INTERFACE ITF_SubSystem

PROPERTY PUBLIC eCondition : SubLevelCondition
GET
END_GET
END_PROPERTY

PROPERTY PUBLIC nErrorID : UDINT
GET
END_GET
END_PROPERTY

END_INTERFACE

(* stored: Version 1.1.0.1, ProductVersion 3.1.4024.12
   Itf ITF_SubSystem: Id {09154105-ab75-48cb-83dd-c703e22f8f7e}
   Property eCondition: Id {07acda04-f4aa-4889-9552-e7c66af85bb5}
   Get Get: Id {0781b1e4-08b5-4f0a-946d-9624d47875cf}
   Property nErrorID: Id {787c5caa-e97a-4517-b512-292dc9fabe96}
   Get Get: Id {e895180c-0fa7-4dfe-acbd-6ae7f98d2cdf} *)
